{attribute 'GeneratedUsingTerminal: EK1100-0000-0018'}
{attribute addProperty BoxType "EK1100-0000-0018"}
{attribute addProperty Id "Term_24_EK1122Term_24_EK1122_39E7B5CB235Term_31_EL3773EL3773_F128CC82184Term_32_EL2258EL2258_E3B260FA508Term_33_EL3164EL3164_B71BFF4244Term_32_EL9011EL9011_D65D3D320"}
{attribute addProperty CRC "3753839588"}
{attribute addProperty Size "971"}
{attribute addProperty Name "Term 23 (EK1100)"}
TYPE Term_23_EK1100_DFBF0BE4 EXTENDS EK1100_1FC0878B :
STRUCT
	{attribute addProperty Name "Term 24 (EK1122)"}
	{attribute addProperty PreviousPort "Term 23 (EK1100) : B"}
	Term_24_EK1122 : Term_24_EK1122_39E7B5CB;
	{attribute addProperty Name "Term 31 (EL3773)"}
	{attribute addProperty PreviousPort "Term 24 (EK1122) : C"}
	Term_31_EL3773 : EL3773_F128CC82;
	{attribute addProperty Name "Term 32 (EL2258)"}
	{attribute addProperty PreviousPort "Term 31 (EL3773) : B"}
	Term_32_EL2258 : EL2258_E3B260FA;
	{attribute addProperty Name "Term 33 (EL3164)"}
	{attribute addProperty PreviousPort "Term 32 (EL2258) : B"}
	Term_33_EL3164 : EL3164_B71BFF42;
	{attribute addProperty Name "Term 32 (EL9011)"}
	{attribute addProperty PreviousPort "Term 33 (EL3164) : B"}
	Term_32_EL9011 : EL9011_D65D3D32;
END_STRUCT
END_TYPE

(* stored: Version 1.2.0.0, ProductVersion 3.1.4024.11
   DUT Term_23_EK1100_DFBF0BE4: Id {c22a1ec6-b851-02c6-1b17-4dd650909ef3} *)
